(* IEC 61131-3 sources: OMJSON/src/Ar/OMJSON, 2 files *)

(* ---- OMJSON.typ ---- *)
(*
 * File: OMJSON.typ
 * Copyright (c) 2023 Loupe
 * https://loupe.team
 *
 * This file is part of OMJSON, licensed under the MIT License.
 *)

TYPE
	JSON_ERR_enum :
		(
		JSON_ERR_INVALIDINPUT := 50000,
		JSON_ERR_MEMALLOC,
		JSON_ERR_MAXLEVELREACHED,
		JSON_ERR_PARSE,
		JSON_ERR_HUH,
		JSON_ERR_CACHEFULLITEMS,
		JSON_ERR_CACHEFULLVARS,
		JSON_ERR_CACHEEMPTY,
		JSON_ERR_MAXITERATIONS,
		JSON_ERR_WS_KEYNOTFOUND,
		JSON_ERR_WS_FRAGMENT,
		JSON_ERR_WS_RSV,
		JSON_ERR_WS_OPCODE,
		JSON_ERR_WS_MASK,
		JSON_ERR_WS_PAYLOADLENGTH,
		JSON_ERR_TCP_FRAGMENT,
		JSON_ERR_TCP_BAD_PACKET,
		JSON_ERR_NO_LICENSE,
		JSON_ERR_WS_MAX_CLIENTS,
		JSON_ERR_WS_INVALID_MAX_CLIENTS,
		JSON_ERR_ACCESSDENIED,
		JSON_ERR_WS_,
		JSON_ERR_
		);
	JSON_ACCESS_enum :
		(
		JSON_ACCESS_NONE := 0,
		JSON_ACCESS_READ,
		JSON_ACCESS_WRITE,
		JSON_ACCESS_READWRITE
		);
	jsonAccessEntry_typ : 	STRUCT
		name : STRING[VAR_STRLEN_NAME]; (*Variable name. Grants access to the variable and everything below it (members, array elements)*)
		access : JSON_ACCESS_enum; (*Access granted to clients*)
	END_STRUCT;
	jsonAccess_typ : 	STRUCT
		pEntries : UDINT; (*Address of an array of jsonAccessEntry_typ. Variables that are not covered by an entry are not accessible*)
		numEntries : UINT; (*Number of elements in the array at pEntries. 0 denies all access*)
		disableWrites : BOOL; (*Reject all writes, regardless of entries*)
		allowedClientIP : ARRAY[0..JSON_MAI_CLIENTS]OF STRING[TCPCOMM_STRLEN_IPADDRESS]; (*Client IP addresses allowed to connect. All empty allows any client*)
		deniedReadCount : UDINT;
		deniedWriteCount : UDINT;
		deniedConnectCount : UDINT;
		lastDeniedName : STRING[VAR_STRLEN_NAME];
		lastDeniedClientIP : STRING[TCPCOMM_STRLEN_IPADDRESS];
	END_STRUCT;
	jsonWSS_client_info_typ : 	STRUCT
		Connected : BOOL;
		TimeSinceLastRequest_ms : UDINT;
		ClientIP : STRING[TCPCOMM_STRLEN_IPADDRESS];
		ClientPort : UINT;
	END_STRUCT;
	jsonWSS_client_debug_typ : 	STRUCT
		socketConnectCount : DINT;
		websocketConnectCount : DINT;
		socketDisconnectCountTimeout : DINT;
		socketDisconnectCountOpcode : DINT;
		socketDisconnectCountError : DINT;
		socketDisconnectCountRecvLength0 : DINT;
		socketInvalidCountError : DINT;
		noDataCount : DINT;
		dataCount : DINT;
		justRightCount : DINT;
		tooBigCount : DINT;
		tooSmallCount : DINT;
		doubleDataCount : DINT;
		oldDataReceived : BOOL;
	END_STRUCT;
	jsonWSServer_int_client_typ : 	STRUCT
		wsStream : WSStream_typ;
		pReceiveData : UDINT;
		pSendData : UDINT;
		messageBuffer : datbufBuffer_typ;
		wsConnected : BOOL;
		writeVariable : jsonWriteVariable;
		readVariableList : jsonReadVariableList;
		debug : jsonWSS_client_debug_typ;
		requestTimer : TON_10ms;
		pCache : REFERENCE TO jsonCache_typ;
	END_STRUCT;
	jsonWSServer_Internal_typ : 	STRUCT
		initialized : BOOL;
		wsServer : WSConnectionManager_typ;
		client : ARRAY[0..JSON_MAI_CLIENTS]OF jsonWSServer_int_client_typ;
		requestTimer : TON_10ms;
		iClient : UINT;
		connectedClients : UINT;
		maxClients : UINT;
	END_STRUCT;
	jsonHTTPServer_Int_Debug_typ : 	STRUCT
		readSendCommand : BOOL;
	END_STRUCT;
	jsonHTTPServer_Int_Write_typ : 	STRUCT
		webService : httpService;
		pUri : UDINT;
		pRequestData : UDINT;
		ResponseHeader : httpResponseHeader_t;
		processed : BOOL;
		writeVariable : jsonWriteVariable;
	END_STRUCT;
	jsonHTTPServer_Int_Read_typ : 	STRUCT
		webService : httpService;
		pUri : UDINT;
		pRequestData : UDINT;
		ResponseHeader : httpResponseHeader_t;
		processed : BOOL;
		readVariableList : jsonReadVariableList;
	END_STRUCT;
	jsonHTTPServer_Internal_typ : 	STRUCT
		initialized : BOOL;
		read : jsonHTTPServer_Int_Read_typ;
		write : jsonHTTPServer_Int_Write_typ;
		debug : jsonHTTPServer_Int_Debug_typ;
	END_STRUCT;
	jsonWSConnect_Internal_typ : 	STRUCT
		encodeBase64 : httpEncodeBase64;
	END_STRUCT;
	JSON_TYPE_enum :
		(
		JSON_TYPE_INVALID := 0,
		JSON_TYPE_OBJECT_ELEMENT,
		JSON_TYPE_ARRAY_ELEMENT
		);
	jsonStructLevel_typ : 	STRUCT
		variable : varVariable_typ;
		iItem : UINT;
		jsonType : JSON_TYPE_enum;
	END_STRUCT;
	jsonWriteVariable_Int_typ : 	STRUCT
		initialized : BOOL;
		pJSONObject : UDINT;
		pChar : UDINT;
		iStructLevel : INT;
		structLevel : ARRAY[0..JSON_MAI_STRUCTLEVEL]OF jsonStructLevel_typ;
	END_STRUCT;
	jsonReadVariableList_Int_typ : 	STRUCT
		initialized : BOOL;
		outputBuffer : datbufBuffer_typ;
		readVariable : jsonReadVariable;
	END_STRUCT;
	jsonReadVariable_Int_typ : 	STRUCT
		initialized : BOOL;
		outputBuffer : datbufBuffer_typ;
		variableName : STRING[VAR_STRLEN_NAME];
		addVariableToCache : jsonAddVariableToCache;
	END_STRUCT;
	jsonAddVariableToCache_Int_typ : 	STRUCT
		initialized : BOOL;
		iStructLevel : INT;
		structLevel : ARRAY[0..JSON_MAI_STRUCTLEVEL]OF jsonStructLevel_typ;
	END_STRUCT;
	jsonCache_typ : 	STRUCT
		iVariable : UINT;
		variable : ARRAY[0..JSON_MAI_CACHEVAR]OF jsonCacheVariable_typ;
		iItem : UINT;
		item : ARRAY[0..JSON_MAI_CACHEITEM]OF jsonCacheItem_typ;
	END_STRUCT;
	jsonCacheVariable_typ : 	STRUCT
		name : STRING[VAR_STRLEN_NAME];
		iStart : UINT;
		iEnd : UINT;
	END_STRUCT;
	jsonCacheItem_typ : 	STRUCT
		prefix : STRING[JSON_STRLEN_PREFIX];
		variable : varVariable_typ;
		suffix : STRING[JSON_STRLEN_SUFFIX];
	END_STRUCT;
	jsonReadVarNoCache_Int_typ : 	STRUCT
		initialized : BOOL;
		outputBuffer : datbufBuffer_typ;
		iStructLevel : INT;
		structLevel : ARRAY[0..JSON_MAI_STRUCTLEVEL]OF jsonStructLevel_typ;
	END_STRUCT;
END_TYPE

(* ---- OMJSON.fun ---- *)
(*
 * File: OMJSON.fun
 * Copyright (c) 2023 Loupe
 * https://loupe.team
 *
 * This file is part of OMJSON, licensed under the MIT License.
 *)

FUNCTION_BLOCK jsonWebSocketServer (*Serve variables via JSON and WebSockets*) (*$GROUP=User*)
	VAR_INPUT
		pCacheArray : UDINT; (*Address of the variable cache array. Number of elements in array needs to be equal to numClients*)
		maxClients : UINT; (*Number of clients supported at a time. 0 defaults to 1*)
		ServerIP : STRING[TCPCOMM_STRLEN_IPADDRESS]; (*IP Address of the server*)
		ServerPort : UINT; (*Port to be used by server*)
		BufferSize : UDINT; (*Size of buffers. N buffers will be allocated, so the total memory requirement is N*BufferSize.*)
		MaxIterations : UDINT; (*Maximum number of iterations for looping through variables.*)
		AcknowledgeError : BOOL; (*Acknowledge errors. Automatically reset by FUB.*)
		Timeout : UDINT; (*Max time in miliseconds since last message from client before forcing disconnect*)
		pAccess : UDINT; (*Optional address of a jsonAccess_typ. 0 allows access to all variables*)
	END_VAR
	VAR_OUTPUT
		ClientInfo : ARRAY[0..JSON_MAI_CLIENTS] OF jsonWSS_client_info_typ;
		AccessControlActive : BOOL; (*An access list is in use. If FALSE, clients can read and write all variables*)
		Error : BOOL;
		ErrorID : UINT;
		ErrorString : STRING[JSON_STRLEN_ERROR];
	END_VAR
	VAR
		internal : jsonWSServer_Internal_typ;
	END_VAR
END_FUNCTION_BLOCK

FUNCTION_BLOCK jsonHTTPServer (*Serve variables via JSON and HTTP*) (*$GROUP=User*)
	VAR_INPUT
		pCache : UDINT; (*Address of the variable cache*)
		ServiceNamePrefix : STRING[JSON_STRLEN_SERVICENAMEPREFIX]; (*Optional service name prefix*)
		BufferSize : UDINT; (*Size of buffers. N buffers will be allocated, so the total memory requirement is N*BufferSize.*)
		MaxIterations : UDINT; (*Maximum number of iterations for looping through variables.*)
		AcknowledgeError : BOOL; (*Acknowledge errors. Automatically reset by FUB.*)
		pAccess : UDINT; (*Optional address of a jsonAccess_typ. 0 allows access to all variables*)
	END_VAR
	VAR_OUTPUT
		AccessControlActive : BOOL; (*An access list is in use. If FALSE, clients can read and write all variables*)
		Error : BOOL;
		ErrorID : UINT;
		ErrorString : STRING[JSON_STRLEN_ERROR];
	END_VAR
	VAR
		internal : jsonHTTPServer_Internal_typ;
	END_VAR
END_FUNCTION_BLOCK

FUNCTION_BLOCK jsonWriteVariable (*Write variable values received as a JSON object*) (*$GROUP=User*)
	VAR_INPUT
		pJSONObject : UDINT; (*Address of the JSON object*)
		MaxJSONObjectLength : UDINT; (*Maximum length of the JSON object*)
		MaxIterations : UDINT; (*Maximum number of iterations for expanding structures*)
		pAccess : UDINT; (*Optional address of a jsonAccess_typ. 0 allows access to all variables*)
	END_VAR
	VAR_OUTPUT
		Status : UINT; (*0 = Done, 65535 = Busy, other values are errors*)
	END_VAR
	VAR
		internal : jsonWriteVariable_Int_typ;
	END_VAR
END_FUNCTION_BLOCK

FUNCTION_BLOCK jsonReadVariableList (*Convert a list of variables into a JSON object*) (*$GROUP=User*)
	VAR_INPUT
		pVariableList : UDINT;
		pCache : UDINT;
		BufferSize : UDINT;
		MaxIterations : UDINT;
		pAccess : UDINT; (*Optional address of a jsonAccess_typ. 0 allows access to all variables*)
	END_VAR
	VAR_OUTPUT
		Status : UINT;
		pJSONObject : UDINT;
		JSONObjectLength : UDINT;
	END_VAR
	VAR
		internal : jsonReadVariableList_Int_typ;
	END_VAR
END_FUNCTION_BLOCK

FUNCTION_BLOCK jsonReadVariable (*Convert a variable into a JSON object*) (*$GROUP=User*)
	VAR_INPUT
		pVariableName : UDINT;
		pCache : UDINT;
		BufferSize : UDINT;
		MaxIterations : UDINT;
		pAccess : UDINT; (*Optional address of a jsonAccess_typ. 0 allows access to all variables*)
	END_VAR
	VAR_OUTPUT
		Status : UINT;
		pJSONObject : UDINT;
		JSONObjectLength : UDINT;
	END_VAR
	VAR
		internal : jsonReadVariable_Int_typ;
	END_VAR
END_FUNCTION_BLOCK

FUNCTION_BLOCK jsonAddVariableToCache (*Add a variable to the JSON variable cache*) (*$GROUP=User*)
	VAR_INPUT
		pVariableName : UDINT;
		pCache : UDINT;
		MaxIterations : UDINT;
	END_VAR
	VAR_OUTPUT
		Status : UINT;
		iVariable : UINT;
	END_VAR
	VAR
		internal : jsonAddVariableToCache_Int_typ;
	END_VAR
END_FUNCTION_BLOCK

FUNCTION_BLOCK jsonReadVariableNoCache (*Convert a variable into a JSON object without caching*) (*$GROUP=User*)
	VAR_INPUT
		pVariableName : UDINT; (*Address of name of variable to convert to JSON*)
		BufferSize : UDINT; (*Size of internal data buffer*)
		MaxIterations : UDINT; (*Maximum number of iterations for expanding structures*)
		pAccess : UDINT; (*Optional address of a jsonAccess_typ. 0 allows access to all variables*)
	END_VAR
	VAR_OUTPUT
		Status : UINT; (*0 = Done, 65535 = Busy, other values are errors*)
		pJSONObject : UDINT; (*Address of the generated JSON object*)
		JSONObjectLength : UDINT; (*Length of the generated JSON object*)
	END_VAR
	VAR
		internal : jsonReadVarNoCache_Int_typ;
	END_VAR
END_FUNCTION_BLOCK

FUNCTION jsonUnescape : UDINT (*Unescape JSON string*)
	VAR_INPUT
		pDest : UDINT;
		pSrc : UDINT;
		maxLength : UDINT;
		reentry : UDINT;
	END_VAR
END_FUNCTION

FUNCTION jsonEscape : UDINT (*Escape JSON string*)
	VAR_INPUT
		pDest : UDINT;
		pSrc : UDINT;
		maxLength : UDINT;
		reentry : UDINT;
	END_VAR
END_FUNCTION
